(* IEC 61131-3 sources: AutomationStudioProjects/Project Maszyny grawerującej/Program, 7 files *)

(* ---- Types.typ ---- *)
TYPE
	ManualStateEnum :
		( (*State in manual work describe if move in axis is able*)
		MANUAL_MOVE_ACTIVE := 0, (*in this state able is move *)
		MANUAL_MOVE_NONACTIVE := 1 (*In this move axis is enable*)
		);
	AxisStateEnum :
		( (*State in main program  decided about axises*)
		STATE_DEFAULT := 0, (*Machine is in this state after  switch on main power*)
		STATE_READY := 1, (*Motors are ready to next action*)
		STATE_HOME := 2, (*In this state motors are hommed, are in "safety" position*)
		STATE_POWER := 3, (*In this state motors are powered on*)
		STATE_MATUAL_WORK := 4, (*Machine is in ManualMode*)
		STATE_AUTO_WORK := 5, (*Machine is in AutoMode*)
		STATE_ESTOP := 6,
		STATE_ERROR := 7 (*Machine has some error*)
		);
	AutoStateEnum :
		( (*State in Auto mode*)
		STATE_WAIT_START := 0, (*Machine wait for activated porocedure *)
		STATE_DRIVE := 1, (*Eelemnt drive to processing place*)
		STATE_MEASUREMENT := 2, (*Element is measured*)
		STATE_POS_AFTER_MES := 3, (*In this state axis X is homed after mesured element*)
		STATE_COMPARE_STRING := 4, (*in this state is compared length of sitrng and element *)
		STATE_GOTO_CENTER := 5, (*Spindle go to center of elements*)
		STATE_HOME_ON_CENTER := 6,
		STATE_ENGRAVING := 7 (*Element is engraved*)
		);
	LettersEnum :
		( (*Enumetated of letters type*)
		i_LETTER := 0,
		I_LETTER := 1,
		R_LETTER := 2,
		U_LETTER := 3,
		W_LETTER := 4,
		X_LETTER := 5
		);
END_TYPE

(* ---- Alarm.st ---- *)
(*********************************************************************************
 * Copyright:
 * Author:    ppiwo
 * Created:   July 27, 2022/10:53 AM
 * Description: In this action is described setting falg which tell about axis is in dangerous position.
 *********************************************************************************)

ACTION actionAlarm:

	(* --- In IF structure is setting flags when position cross some value --- *)
	IF AxisState  = STATE_MATUAL_WORK THEN

		(* --- Setting value of flag dependent on positon Axis Z --- *)
		IF MpCnc3Axis_0.Z > 295 THEN
			FlagDisableJogPos		:= TRUE;
		ELSE
			FlagDisableJogPos		:= FALSE;
		END_IF;

		IF MpCnc3Axis_0.Z < 5 THEN
			FlagDisableJogNeg		:= TRUE;
		ELSE
			FlagDisableJogNeg		:= FALSE;
		END_IF;

		(* --- Setting value of flag dependent on positon Axis Y --- *)
		IF MpCnc3Axis_0.Y > 245 THEN
			FlagDisableJogPosY		:= TRUE;
		ELSE
			FlagDisableJogPosY		:= FALSE;
		END_IF;

		IF MpCnc3Axis_0.Y < -245 THEN
			FlagDisableJogNegY		:= TRUE;
		ELSE
			FlagDisableJogNegY		:= FALSE;
		END_IF;
	END_IF;

END_ACTION

(* ---- AutoWork.st ---- *)
(*********************************************************************************
 * Copyright:
 * Author:    ppiwo
 * Created:   July 12, 2022/11:00 AM
 * Description: In this file is located logic of Finite State Machine
				which supports automaticly engraving of elements.
 *********************************************************************************)

ACTION actionAutoWork:

	(* --- Condition to go to ManualMode ---
			Machine can go to ManualMode in all AutoState except Engraving state *)
	IF (AutoState <> STATE_ENGRAVING) AND (SwitchManual = TRUE) THEN
		AxisState 									:= STATE_MATUAL_WORK;
	END_IF;

	(* --- Finite State Machine described working machine in Auto mode --- *)
	CASE AutoState OF

		(* STATE_WAIT_START is default state when machine go to Auto mode.
			In this state machine wait for signal from switchStart (clicked in visualization)
			and go to STATE_DRIVE. *)
		STATE_WAIT_START:
			(* Set Flag to corecr value to have corret action of AutoMode. Set new parameters of axis. *)
			FlagAbleSet 							:= TRUE;
			FlagDisableConfMove						:= TRUE;
			actionSetAxisParameters;
			MpAxisBasic_X.Update					:= TRUE;

			IF SwitchStart = TRUE THEN
				AutoState 							:= STATE_DRIVE;
			END_IF;
			IF PowerOnSwitch = FALSE THEN
				AxisState							:= STATE_DEFAULT;
			END_IF
			(* STATE_DRIVE is state where element commute to processing place.
				Element drive with high speed and when element enter to processing area (laser sensor give high level)
				speed is set a low speed to make better accuracy.
				In this state memorized value of position when object is firstly detected and FSM go to nest state.   *)
		STATE_DRIVE:
			MpAlarmXReset(gAlarmXCore,'Too short object');	//Reset alarm
			MpCnc3Axis_0.MoveProgram				:= FALSE;
			FlagDisableConfMove						:= TRUE;
			(* --- reset value of measure temp variable --- *)
			startMeasurePos							:= 0;
			endMeasurePos							:= 0;

			(* --- logic of drive --- *)
			AxisParameters[0].Velocity 				:= XVelFast;
			MpAxisBasic_X.MoveVelocity				:= TRUE;

			IF diLaserSensor = TRUE AND prevLaserSensorState = FALSE THEN
				startMeasurePos 					:= LREAL_TO_REAL(MpCnc3Axis_0.X);
				AxisParameters[0].Velocity 			:= XVelSlow;
				MpAxisBasic_X.Update 				:= TRUE;
				prevLaserSensorState				:= diLaserSensor;
				AutoState							:= STATE_MEASUREMENT;
			END_IF;

			ChosenLetter							:= RemembLetter; //Update value of ChosenLetter

			(* IN this sate element is measure. Position when element is not in processing area is memorized in variable.
			length of element is diffrence between start and end position.
			After measure axis X is stopped and FSM go to state homing on front of element.  *)
		STATE_MEASUREMENT:
			IF  diLaserSensor = FALSE AND prevLaserSensorState = TRUE THEN
				endMeasurePos						:= LREAL_TO_REAL(MpCnc3Axis_0.X);
				LenghtOfElement						:= ABS(startMeasurePos-endMeasurePos);
				MpAxisBasic_X.MoveVelocity			:= FALSE;
				prevLaserSensorState				:= diLaserSensor;
				AutoState							:= STATE_POS_AFTER_MES;
			END_IF;

			(* In this state axis X is homing in front of element.
			 at first axis go to front of element and set move to false. When move is false axis is homed
			After homing FSM go to next state. *)
		STATE_POS_AFTER_MES:
			AxisParameters[0].Position 				:= endMeasurePos;
			MpAxisBasic_X.Update					:= TRUE;
			MpAxisBasic_X.MoveAbsolute				:= TRUE;
			AutoState								:= STATE_COMPARE_STRING;

			(* In is compare length of string with length of elemnt.
			Length of string saved in constant variable and is chosen by structue CASE.
			To length of string is added 40[mm] because engraving is made 20mm from the all edge.
			If length of string if greater than len of elements we have error in other case go to next state. *)
		STATE_COMPARE_STRING:
			LenOfString								:= 0;
			MpAxisBasic_X.MoveAbsolute				:= FALSE;
			CASE ChosenLetter OF
				i_LETTER:
					LenOfString						:= LEN_i;
				I_LETTER:
					LenOfString						:= LEN_I;
				R_LETTER:
					LenOfString						:= LEN_R;
				U_LETTER:
					LenOfString						:= LEN_U;
				W_LETTER:
					LenOfString						:= LEN_W;
				X_LETTER:
					LenOfString						:= LEN_X;
			END_CASE;

			LenOfString								:= LenOfString + 40;

			IF LenOfString <= LenghtOfElement THEN
				AutoState							:= STATE_GOTO_CENTER;

			ELSE
				MpAlarmXSet(gAlarmXCore,'Too short object');
				showMesBox							:= TRUE; 	//set flag to show messege box with text about that object is too short
				AutoState							:= STATE_DRIVE;

			END_IF;

			(* In this state axis X go to  center of element.
			Center of element is calculated by mean and go to this point by additive move.
			When axis is in position move is switched off and FSM go to next state.  *)
		STATE_GOTO_CENTER:
			CenterOfElement							:= LenghtOfElement / 2;
			AxisParameters[0].Distance 				:= - CenterOfElement;
			MpAxisBasic_X.Update					:= TRUE;
			MpAxisBasic_X.MoveAdditive				:= TRUE;
			IF MpAxisBasic_X.MoveDone = TRUE THEN
				MpAxisBasic_X.MoveAdditive			:= FALSE;
				AutoState							:= STATE_HOME_ON_CENTER;
			END_IF;

		(* In this state axis X is homing in center of element.
			When motor is homed FSM go to next step*)
		STATE_HOME_ON_CENTER:
			MpAxisBasic_X.Home						:= TRUE;

			(* --- condition to step to next state ---
				I made condition with direct position and flag ComandBusy to have
				confidence that axis is homed  *)
			IF MpCnc3Axis_0.X = 0 AND MpAxisBasic_X.CommandBusy = FALSE THEN
				MpAxisBasic_X.Home					:= FALSE;
				AutoState							:= STATE_ENGRAVING;
			END_IF;

		STATE_ENGRAVING:
			//CncParameters.MoveProgramOptions.StartMode:=mcPRGSM_SIMULATION_GEOMETRY;
			CASE ChosenLetter OF
				i_LETTER:
					CncParameters.ProgramName 		:= 'LetterSi';
				I_LETTER:
					CncParameters.ProgramName 		:= 'LetterI';
				W_LETTER:
					CncParameters.ProgramName 		:= 'LetterW';
				R_LETTER:
					CncParameters.ProgramName 		:= 'LetterR';
				X_LETTER:
					CncParameters.ProgramName 		:= 'LetterX';
				U_LETTER:
					CncParameters.ProgramName 		:= 'LetterU';

			END_CASE;
			(* --- remember press switch STOPProgram when object is envraving --- *)
			IF SwitchStop=TRUE THEN
				RememberStop						:= TRUE;
			END_IF;

			MpCnc3Axis_0.MoveProgram				:= TRUE;

			(* --- Check if pozition on axis Z is 99 ---
					use it ro M-Function*)
			IF MpCnc3Axis_0.Z > 100 THEN
				EngravingLevel						:= FALSE;
			ELSE
				EngravingLevelUp					:= FALSE;
			END_IF;

			IF MpCnc3Axis_0.MoveDone = TRUE THEN
				FlagDisableConfMove					:= FALSE;
				AutoState							:= STATE_DRIVE;
			END_IF;

	END_CASE;

	(* --- Stop AutoMode ---
			AutoMode is stopping when object is not engraving.
			When STOP was pressed in state ENGRAVING, program was doing to end and AutoMode is stopped. *)
	IF AutoState <> STATE_ENGRAVING THEN
		IF (RememberStop = TRUE) OR (SwitchStop = TRUE) THEN
			MpAxisBasic_X.MoveVelocity				:= FALSE;
			RememberStop							:= FALSE;
			AutoState								:= STATE_WAIT_START;
		END_IF;
	END_IF;
END_ACTION

(* ---- Main.st ---- *)
(*********************************************************************************
 * Copyright:
 * Author:    ppiwo
 * Created:   July 11, 2022/1:00 PM
 * Description: File with Fine State Machine of homing motors and configuration of used motors
 *********************************************************************************)

PROGRAM _INIT
    (*--- Enable MpCnc3Axis ---
		Enable MpCncsAxis and define parameters*)
	MpCnc3Axis_0.Enable 				:= TRUE;
	MpCnc3Axis_0.Override 				:= 100.0;
	CncParameters.ProgramName 			:= 'GoToHome';

	(*--- Enable MpAxisBasic ---
		Enable MpAxisBasic and define parameters*)
	MpAxisBasic_X.Enable				:= TRUE;
	MpAxisBasic_Y.Enable 				:= TRUE;
	MpAxisBasic_Z.Enable 				:= TRUE;
	MpAxisSpindle.Enable 				:= TRUE;

	(* --- Set default Axis Parameters --- *)
	actionSetAxisParameters;

	(* --- Initialize value of variables in program ---  *)
	diEmergencyStop						:= TRUE; //Set high level Emergency Stop to have confidence thet in HMI it has value TRUE
	PathPrevStatus						:= 0;
	svg_path 							:= '/FileDevice:CNC_ProgDir/PathPreview.svg'; //Initialize path to draw trajectory
	svg_string;
	FlagEstop							:= FALSE;

	(* --- Set enable and MpLink of Alarm Core and AlarmHistoryCore --- *)
	AlarmCore.MpLink					:= ADR(gAlarmXCore);
	AlarmCore.Enable					:= TRUE;

	AlarmHistoryCore.MpLink				:= ADR(gAlarmXHistory);
	AlarmHistoryCore.Enable				:= TRUE;

END_PROGRAM

PROGRAM _CYCLIC

(* --- Initialize of AlarmCore and AlarmHistoryCore --- *)
	AlarmCore();
	AlarmHistoryCore();

(* --- Initialize MpCncAxis and all MpAxisBasic ---
	  Initialize axis by before prepered parameters  in Init Block*)

	MpCnc3Axis_0.MpLink 				:= ADR(gCncXYZ);
	MpCnc3Axis_0.Parameters 			:= ADR(CncParameters);
	MpCnc3Axis_0();
	MpAxisBasic_X.MpLink     			:= ADR(gAxisQX);
	MpAxisBasic_X.Parameters 			:= ADR(AxisParameters[0]);
	MpAxisBasic_X();
	MpAxisBasic_Y.MpLink    			:= ADR(gAxisQY);
	MpAxisBasic_Y.Parameters 			:= ADR(AxisParameters[1]);
	MpAxisBasic_Y();
	MpAxisBasic_Z.MpLink     			:= ADR(gAxisQZ);
	MpAxisBasic_Z.Parameters 			:= ADR(AxisParameters[2]);
	MpAxisBasic_Z();
	MpAxisSpindle.MpLink     			:= ADR(gAxisQS);
	MpAxisSpindle.Parameters 			:= ADR(AxisParameters[3]);
	MpAxisSpindle();

	actionAlarm; // Check position Z, Y position and set flag to alarm/enable switch JOG

	(* --- Transition to STATE_ERROR ---*)
	IF MpCnc3Axis_0.Error THEN
		AxisState							:= STATE_ERROR;
	END_IF;

	(* --- Service press Emenrency STOP ---
			Motors of machine are switch off and machine go to STATE_DEFAULT,
			AutoMOde goto STATE_WAIT_START*)
	IF diEmergencyStop = FALSE THEN
		MpCnc3Axis_0.Stop				:= TRUE;
		FlagPresEStop 					:= TRUE;
		AxisState 						:= STATE_DEFAULT;
		AutoState 						:= STATE_WAIT_START;
	END_IF;

	(*--- Finite State Machine to powered on and homed motors ---*)
	CASE AxisState OF

		(* In STATE_DEFAULT machine is automaticly after switch on main power. In this state all axis action is reset
			FSM go to next state when PowerOnSwitch is on high level and Flag ReadyToPowerOn is true *)
		STATE_DEFAULT:

			(* Reset all parameters of motors  *)
			MpCnc3Axis_0.Stop			:= FALSE;
			MpCnc3Axis_0.Power			:= FALSE;
			MpCnc3Axis_0.Home			:= FALSE;
			MpCnc3Axis_0.MoveProgram	:= FALSE;

			MpAxisBasic_X.MoveAbsolute	:= FALSE;
			MpAxisBasic_X.MoveAdditive	:= FALSE;
			MpAxisBasic_X.MoveVelocity	:= FALSE;

			ConfXPos					:= FALSE;
			ConfYPos					:= FALSE;
			ConfZPos					:= FALSE;

			FlagAbleSet					:= TRUE;
			FlagConfirmError 			:= FALSE;
			MpAlarmXReset(gAlarmXCore,'Axis Error');

			(* Set new Axis Parameters *)
			actionSetAxisParameters;

			IF PowerOnSwitch = TRUE AND MpCnc3Axis_0.Info.ReadyToPowerOn = TRUE  THEN //transition to StatePower
				AxisState				:= STATE_POWER;
			END_IF;

			(* In STATE_POWER all axis are powerd on, when flag PowerOn is in high level FSM go to nest step *)
		STATE_POWER:

			MpCnc3Axis_0.Power			:= TRUE; //motors are powered on

			IF MpCnc3Axis_0.PowerOn = TRUE THEN  //Transition to StateHome, check if motors is powered on
				AxisState				:= STATE_HOME;
			END_IF;

			(* In STATE_HOME all axis is homed. We set up taht in the first time machine is in safety position.
			    Next step is able if flag IsHomed is True. If machine is switch on after EStop axis Y and Z go to homing position *)
		STATE_HOME:
			IF (FlagPresEStop = FALSE)  THEN
				MpCnc3Axis_0.Home		:= TRUE; //Motors are homed
				IF MpCnc3Axis_0.IsHomed = TRUE THEN //Transition to StateReady, check if motors is homed on
					AxisState			:= STATE_READY;
				END_IF;
			ELSE
				(* Service case when Emergency STOP was used *)
				IF FlagEstop = TRUE THEN
					CncParameters.ProgramName	:= 'GoToHome';
					MpCnc3Axis_0.MoveProgram	:= TRUE;
					IF MpCnc3Axis_0.MoveDone = TRUE THEN
						FlagPresEStop			:= FALSE;
						MpCnc3Axis_0.MoveProgram:= FALSE;
						FlagEstop       		:= FALSE;
						AxisState				:= STATE_READY;
					END_IF;
				END_IF;
			END_IF;

			(* STATE_READY is  state when machine could start workin with element.
				This state have 2 substeps, which are mode of work machine *)
		STATE_READY:
			MpCnc3Axis_0.Home			:= FALSE;
			IF SwitchAuto THEN
				AxisState 				:= STATE_AUTO_WORK;
			END_IF;

			IF SwitchManual THEN
				AxisState 				:= STATE_MATUAL_WORK;
			END_IF;

			(* In this  state machine work in Automatic mode.
				Machine in Auto mode drive to processing place, measure elements and engraving elements  *)
		STATE_AUTO_WORK:
			actionAutoWork;

			(* In this  state machine work in Manualy mode.
				Operator make all activity to move machine and engraving elements  *)
		STATE_MATUAL_WORK:
			actionSetAxisParameters;
			actionManualWork;

			(* In this state is described behavior when machine has some errors.
			   When error is detected machine is stopping and is setting alarm.
			   If Alarm is confirmed error is deleted and machine return into STATE_DEFAULT*)
		STATE_ERROR:
			(* Motors are off *)
			MpCnc3Axis_0.Power			:= FALSE;
			MpCnc3Axis_0.Home			:= FALSE;
			MpCnc3Axis_0.MoveProgram	:= FALSE;
			MpAlarmXSet(gAlarmXCore,'Axis Error');

			IF FlagConfirmError = TRUE THEN
				MpCnc3Axis_0.ErrorReset		:= TRUE;
			END_IF;
			IF  NOT MpCnc3Axis_0.Error THEN //transition to go out from stateError
				MpCnc3Axis_0.ErrorReset	:= FALSE;
				AxisState				:= STATE_DEFAULT;
			END_IF;
	END_CASE;

	(* Rewriting value od sensor to physical output *)
	IF diLaserSensor=TRUE THEN
		doLaserSensor:=TRUE;
	ELSE
		doLaserSensor:=FALSE;
	END_IF;
END_PROGRAM

PROGRAM _EXIT
	MpCnc3Axis_0(Enable := FALSE);
END_PROGRAM

(* ---- ManualWork.st ---- *)
(*********************************************************************************
 * Copyright:
 * Author:    ppiwo
 * Created:   July 19, 2022/10:35 AM
 * Description: In this action is describing functionality of ManualMode.
				In ManualMode is applied move to set position with set velocity.
				Moreover in this mode is applied Jog mode and switch on spindle with set velocity
 *********************************************************************************)

ACTION actionManualWork:

(* --- Reset before activeted move and set all necessery parameters to basic value *)
	(* Set to basic parameters of single axis *)
	MpAxisBasic_X.MoveVelocity					:= FALSE;
	AxisParameters[0].Velocity 					:= 0;
	AxisParameters[1].Velocity 					:= 0;
	AxisParameters[2].Velocity 					:= 0;
	AxisParameters[3].Velocity 					:= 0;
	MpAxisBasic_X.Update						:= TRUE;
	(* Set AutoState to basic value *)
	AutoState 									:= STATE_WAIT_START;
	FlagDisableConfMove							:= FALSE;
	(* --- Set parameters of Jog move --- *)

(* --- Set flag, witch tell when able next move in ManualMode ---
		This flag is used to blocing or unblocking next move, like said in specification taht in ManualMode we
		can move once axis plus spindle. This flag is in high level when all (3) Cnc axis don't move, next move will be realized.
		When Flag is in high level albe is to change mode to AutoMode an able is switch off the machine.  *)
	IF MpAxisBasic_X.MoveActive = FALSE AND MpAxisBasic_Y.MoveActive = FALSE
		AND MpAxisBasic_Z.MoveActive = FALSE  THEN
		FlagAbleSet								:= TRUE;
		IF PowerOnSwitch = FALSE THEN
			AxisState							:= STATE_DEFAULT;
		END_IF
		IF SwitchAuto THEN
			AxisState							:=STATE_AUTO_WORK;
		END_IF;
	ELSE
		FlagAbleSet								:= FALSE;
		;
	END_IF;

(* --- Main Logic of ManualMode ---
		In case is decided which axis will be moved
		in IF with SwitchSpindelOnOff is decidec if spindle will be actived Spindel could be active parallel with other axis *)
	IF SwitchSpindleOnOff = TRUE THEN
		AxisParameters[3].Velocity				:= SpindleVelocityIn;
		MpAxisSpindle.MoveVelocity				:= TRUE;
	ELSE
		AxisParameters[3].Velocity				:= 0;
		MpAxisSpindle.Update					:= TRUE;
		MpAxisSpindle.MoveVelocity				:= FALSE;

	END_IF;

	CASE ManualState OF
		MANUAL_MOVE_NONACTIVE:
			IF FlagAbleSet = TRUE THEN
	  			ManualState						:= MANUAL_MOVE_ACTIVE;
			END_IF;
		MANUAL_MOVE_ACTIVE:

			(* --- Move to set position ---
			If some axis is set to move, value of position and velocity in this axis is updated and realized move.
			After move switches of confirmation are reset to allow next move.
			Unfortunately this structure doesn't protect to rememberd setting parameters in previous terms, like X axis *)
			IF ConfXPos = TRUE THEN
				AxisParameters[0].Position 			:= XPosition;
				AxisParameters[0].Velocity 			:= XVelocity;
				MpAxisBasic_X.Update				:= TRUE;
				MpAxisBasic_X.MoveAbsolute 			:= TRUE;
				IF MpAxisBasic_X.MoveDone = TRUE THEN
					ConfXPos 						:= FALSE;
					ConfYPos 						:= FALSE;
					ConfZPos 						:= FALSE;
					MpAxisBasic_X.MoveAbsolute 		:= FALSE;
				END_IF;

			ELSIF ConfYPos = TRUE THEN
				AxisParameters[1].Position 			:= YPosition;
				AxisParameters[1].Velocity 			:= YVelocity;
				MpAxisBasic_X.Update				:= TRUE;
				MpAxisBasic_Y.MoveAbsolute 			:= TRUE;
				IF MpAxisBasic_Y.MoveDone = TRUE THEN
					ConfXPos 						:= FALSE;
					ConfYPos 						:= FALSE;
					ConfZPos 						:= FALSE;
					MpAxisBasic_Y.MoveAbsolute 		:= FALSE;
				END_IF;

			ELSIF ConfZPos = TRUE THEN
				AxisParameters[2].Position 			:= ZPosition;
				AxisParameters[2].Velocity 			:= ZVelocity;
				MpAxisBasic_X.Update				:= TRUE;
				MpAxisBasic_Z.MoveAbsolute 			:= TRUE;
				IF MpAxisBasic_Z.MoveDone = TRUE THEN
					ConfXPos 						:= FALSE;
					ConfYPos 						:= FALSE;
					ConfZPos 						:= FALSE;
					MpAxisBasic_Z.MoveAbsolute 		:= FALSE;
				END_IF;

		(* --- Jog move ---
				If button responsible for jog in some axis is activ,
				 jog in this axis is realized *)
			ELSIF JogPlusXActive = TRUE THEN
				MpAxisBasic_X.JogPositive			:= TRUE;

			ELSIF JogMinusXActive = TRUE THEN
				MpAxisBasic_X.JogNegative			:= TRUE;

			ELSIF JogPlusYActive = TRUE THEN
				MpAxisBasic_Y.JogPositive			:= TRUE;

			ELSIF JogMinusYActive = TRUE THEN
				MpAxisBasic_Y.JogNegative			:= TRUE;

			ELSIF JogPlusZActive = TRUE THEN
				MpAxisBasic_Z.JogPositive			:= TRUE;

			ELSIF JogMinusZActive = TRUE THEN
				MpAxisBasic_Z.JogNegative			:= TRUE;
			ELSE
				MpAxisBasic_X.JogPositive			:= FALSE;
				MpAxisBasic_X.JogNegative			:= FALSE;
				MpAxisBasic_Y.JogPositive			:= FALSE;
				MpAxisBasic_Y.JogNegative			:= FALSE;
				MpAxisBasic_Z.JogPositive			:= FALSE;
				MpAxisBasic_Z.JogNegative			:= FALSE;
				ManualState							:= MANUAL_MOVE_NONACTIVE;
			END_IF;
	END_CASE;
END_ACTION

(* ---- SetAxisParameters.st ---- *)
(*********************************************************************************
 * Copyright:
 * Author:    ppiwo
 * Created:   July 27, 2022/10:49 AM
 * Description:In this action is described setting parameters of all Axis like
				velocity, position,acceleration or deceleration.
				Make it in action safe space in main code  and
				improve transparency.
 *********************************************************************************)

ACTION actionSetAxisParameters:
	(* --- Set parameters to axis X --- *)
	AxisParameters[0].Position 			:= 100.0;
	AxisParameters[0].Distance 			:= 360.0;
	AxisParameters[0].Velocity 			:= XVelFast;
	AxisParameters[0].Acceleration 		:= XAcceleration;
	AxisParameters[0].Deceleration 		:= XDecleration;

	(* --- Set parameters to axis Y --- *)
	AxisParameters[1].Position 			:= 100.0;
	AxisParameters[1].Distance 			:= 360.0;
	AxisParameters[1].Velocity 			:= YVel;
	AxisParameters[1].Acceleration 		:= YAcceleration;
	AxisParameters[1].Deceleration 		:= YDecleration;

	(* --- Set parameters to axis Z --- *)
	AxisParameters[2].Position 			:= 100.0;
	AxisParameters[2].Distance 			:= 360.0;
	AxisParameters[2].Velocity 			:= ZVel;
	AxisParameters[2].Acceleration 		:= ZAcceleration;
	AxisParameters[2].Deceleration 		:= ZDecleration;
	AxisParameters[2].Homing.Mode		:= mcHOMING_DEFAULT;

	(* --- Set parameters to Spindle --- *)
	AxisParameters[3].Velocity 			:= 10000.0;
	AxisParameters[3].Acceleration 		:= 10000.0;
	AxisParameters[3].Deceleration 		:= 1000.0;

	(* --- Set Parameters of JOG Mode to axis X --- *)
	CncParameters.Jog.Velocity[0]		:= X_JOG_CNC_VEL;
	AxisParameters[0].Jog.Acceleration	:= XJogAcc;
	AxisParameters[0].Jog.Deceleration	:= XJogDec;
	AxisParameters[0].Jog.Velocity		:= XJogVel;

	(* --- Set Parameters of JOG Mode to axis Y --- *)
	CncParameters.Jog.Velocity[1]		:= Y_JOG_CNC_VEL;
	AxisParameters[1].Jog.Acceleration	:= YJogAcc;
	AxisParameters[1].Jog.Deceleration	:= YJogDec;
	AxisParameters[1].Jog.Velocity		:= YJogVel;

	(* --- Set Parameters of JOG Mode to axis Z --- *)
	CncParameters.Jog.Velocity[2]		:= Z_JOG_CNC_VEL;
	AxisParameters[2].Jog.Acceleration	:= ZJogAcc;
	AxisParameters[2].Jog.Deceleration	:= ZJogDec;
	AxisParameters[2].Jog.Velocity		:= ZJogVel;

	(* --- Call variable CNC program to reseve mamory to their --- *)
	SPINDLE_SPEED;
	FeedFast;
	FeedSlow;
END_ACTION

(* ---- Variables.var ---- *)
(* Variabels nesessery to supports AxisBasic.*)
VAR
	MpAxisBasic_Z : MpAxisBasic; (*Object  describe Axis Z *)
	MpAxisBasic_X : MpAxisBasic; (*Object  describe Axis X*)
	MpAxisBasic_Y : MpAxisBasic; (*Object  describe Axis Y*)
	MpAxisSpindle : MpAxisBasic; (*Object  describe Axis Spindle*)
	AxisParameters : ARRAY[0..3] OF MpAxisBasicParType; (*Instance agregate parameters of  all single axis*)
END_VAR
(* Variabels nesessery to supports CNCAxis.*)
VAR
	MpCnc3Axis_0 : MpCnc3Axis; (*Object  describe CNC Axis*)
	CncParameters : MpCnc3AxisParType; (*Instance agregate parameters of  CNC axis*)
END_VAR
(*Main Variables used in main *)
VAR
	AlarmCore : MpAlarmXCore; (*Object  describe AlarmX*)
	AxisState : AxisStateEnum; (*Variable representet of state machine*)
	PowerOnSwitch : BOOL; (*Variable conected with toggle button which switch on/off motors*)
END_VAR
(*Variables I/O*)
VAR
	prevLaserSensorState : BOOL; (*prev value of laser sensor*)
	diEmergencyStop : BOOL; (*Emergency Stop Button*)
	diLaserSensor : BOOL; (*Variable phisicaly conentet with input, represented laser sensor*)
	doLaserSensor : BOOL; (*Variable phisicaly conentet with output, represented state of laser sensor*)
END_VAR
(*Variables used in main /Used for visualization*)
VAR
	SwitchManual : BOOL; (*Switch mode Manual*)
	SwitchAuto : BOOL; (*Switch mode Auto*)
END_VAR
(*Variabels used in Auto mode / used for visualiztion*)
VAR
	AutoState : AutoStateEnum; (*Variable representet of state AutoMode*)
	SwitchStop : BOOL; (*Stop automatic process*)
	SwitchStart : BOOL; (*Start automatic process*)
	endMeasurePos : REAL; (*Temp variavle to save position in xX axis when enden measure*)
	startMeasurePos : REAL; (*Temp variable to save position in X axis when started measure*)
	LenghtOfElement : REAL; (*Calculated length of element*)
	LenOfString : USINT; (*Calculated length of string*)
	CenterOfElement : REAL; (*Calculated center of element*)
	RemembLetter : LettersEnum; (*Variable representet chosen letter in visualisation*)
	EngravingLevel : BOOL; (*Flag tell than spindel is upper than 100 mm*)
	EngravingLevelUp : BOOL; (*Flag tell than spindel is lower than 100 mm*)
	RememberStop : BOOL; (*Variable which remember press stop when object was engraving*)
	ChosenLetter : LettersEnum; (*chosen letter in visualization update in oyher state than engraving*)
END_VAR
(**)
(*Variabels used inn Manual Mode*)
VAR
	ManualState : ManualStateEnum;
	XPosition : LREAL; (*Value of set position on X axis*)
	XVelocity : REAL; (*Value of velocity in axis X*)
	ConfXPos : BOOL; (*Confirmation of X Pos*)
	YPosition : LREAL; (*Value of set position on Y axis*)
	YVelocity : REAL; (*Value of velocity in axis Y*)
	ConfYPos : BOOL; (*Confirmation of Y Pos*)
	ZPosition : LREAL; (*Value of set position Z axis*)
	ZVelocity : REAL; (*Value of velocity in axis Z*)
	ConfZPos : BOOL; (*Confirm of Z Pos*)
	JogPlusXActive : BOOL; (*Move Jog positive in axis X is enable*)
	JogMinusXActive : BOOL; (*Move Jog negative in axis X is enable*)
	JogPlusYActive : BOOL; (*Move Jog positive in axis Y is enable*)
	JogMinusYActive : BOOL; (*Move Jog negative in axis Y is enable*)
	JogPlusZActive : BOOL; (*Move Jog positive in axis Z is enable*)
	SwitchSpindleOnOff : BOOL; (*switch enabled move spindle axis*)
	JogMinusZActive : BOOL; (*Move Jog negative in axis Z is enable*)
	SpindleVelocityIn : REAL; (*Value of rotation speed of spindle*)
END_VAR
(*Predefinited length of letter*)
VAR CONSTANT
	LEN_I : USINT := 1;
	LEN_i : USINT := 1;
	LEN_W : USINT := 100;
	LEN_R : USINT := 50;
	LEN_U : USINT := 75;
	LEN_X : USINT := 75;
END_VAR
(*Insert your comment here.*)
VAR
	showMesBox : BOOL; (*variable activate messege box in visu when object is too short*)
	FlagDisableConfMove : BOOL; (*Flag switch off enable of move confirm button when machine in auto mode*)
	FlagConfirmError : BOOL := FALSE; (*Flag detect confirm Error stop*)
	FlagEstop : BOOL; (*Flag detect press Emergency stop*)
	FlagPresEStop : BOOL; (*Flag detect if  Emergrncy stop is actual press*)
	FlagAbleSet : BOOL; (*This Flag say us that we can set new position and velocity parameters*)
	FlagDisableJogPos : BOOL; (*flag dialbe a switch JOG*)
	FlagDisableJogNeg : BOOL; (*flag dialbe a switch JOG*)
	FlagDisableJogPosY : BOOL; (*flag dialbe a switch JOG*)
	FlagDisableJogNegY : BOOL; (*flag dialbe a switch JOG*)
END_VAR
(*Value Parameters of  Axis  X*)
VAR
	XVelFast : REAL := 10; (*Value of X fast velocity*)
	XDecleration : REAL := 25; (*Value of deceleration*)
	XAcceleration : REAL := 25; (*Value of acceleration*)
END_VAR
VAR CONSTANT
	X_JOG_CNC_VEL : REAL := 10; (*Value of jog velocity in cnc parameters*)
END_VAR
VAR
	XJogDec : REAL := 5; (*value of jog deceleration*)
	XJogAcc : REAL := 25; (*Value of jog acceleration*)
	XJogVel : REAL := 2; (*Value of jog velocity*)
	XVelSlow : REAL := 5; (*Value of X slow velocity*)
END_VAR
(*Value Parameters of  Axis  Y*)
VAR
	YVel : REAL := 10; (*Value of velocity*)
END_VAR
VAR CONSTANT
	Y_JOG_CNC_VEL : REAL := 10; (*Value of jog velocity in cnc parameters*)
END_VAR
VAR
	YDecleration : REAL := 25; (*Value of deceleration*)
	YJogDec : REAL := 5; (*value of jog deceleration*)
	YJogAcc : REAL := 25; (*Value of jog acceleration*)
	YAcceleration : REAL := 25; (*Value of acceleration*)
	YJogVel : REAL := 2; (*Value of jog velocity*)
END_VAR
(*Value Parameters of  Axis  Z*)
VAR CONSTANT
	Z_JOG_CNC_VEL : REAL := 10; (*Value of jog velocity in cnc parameters*)
END_VAR
VAR
	ZDecleration : REAL := 25; (*Value of deceleration*)
	ZJogDec : REAL := 5; (*value of jog deceleration*)
	ZJogAcc : REAL := 25; (*Value of jog acceleration*)
	ZAcceleration : REAL := 25; (*Value of acceleration*)
	ZJogVel : REAL := 2; (*Value of jog velocity*)
	ZVel : REAL := 10; (*Value of velocity*)
END_VAR
(*Parameters of  CNC program*)
VAR
	FeedSlow : UDINT := 600; (*Slow feed set when letter is engraving*)
	FeedFast : UDINT := 1000; (*Fast feed set when go from/to home position*)
	SPINDLE_SPEED : UDINT := 5000; (*value of spindle speed*)
END_VAR
